ABB RAPID module: MainModule.mod

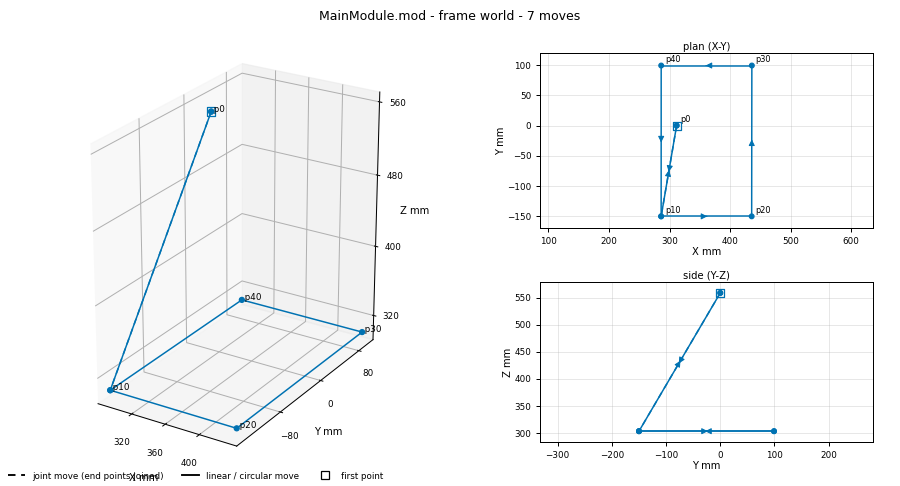
[picture p0: tool path of MainModule.mod in frame world, 7 of 7 moves have a stored position in this frame; points joined in program order, loops and branches not executed]
MODULE MainModule
	CONST robtarget Algus:=[[364.35,0.00,594.00],[0.5,0,0.866025,0],[0,0,0,0],[9E+09,9E+09,9E+09,9E+09,9E+09,9E+09]];
	CONST robtarget p0:=[[311.72,0.00,558.66],[0.0676669,0,0.997708,0],[0,0,0,0],[9E+09,9E+09,9E+09,9E+09,9E+09,9E+09]];
	CONST robtarget p10:=[[286.16,-149.99,303.57],[0.0676667,2.70246E-08,0.997708,1.73496E-07],[-1,0,-1,0],[9E+09,9E+09,9E+09,9E+09,9E+09,9E+09]];
	CONST robtarget p20:=[[435.71,-149.99,303.57],[0.0676665,-1.48195E-07,0.997708,2.84887E-07],[-1,0,-1,0],[9E+09,9E+09,9E+09,9E+09,9E+09,9E+09]];
	CONST robtarget p30:=[[436.00,99.19,303.57],[0.0676668,-2.22625E-07,0.997708,3.78004E-07],[0,-1,0,0],[9E+09,9E+09,9E+09,9E+09,9E+09,9E+09]];
	CONST robtarget p40:=[[286.22,99.19,303.57],[0.0676666,-3.60648E-07,0.997708,3.05387E-07],[0,-1,0,0],[9E+09,9E+09,9E+09,9E+09,9E+09,9E+09]];
	CONST robtarget p50:=[[286.22,99.19,303.57],[0.0676666,-3.60648E-07,0.997708,3.05387E-07],[0,-1,0,0],[9E+09,9E+09,9E+09,9E+09,9E+09,9E+09]];
	TASK PERS tooldata pneumo1:=[TRUE,[[0,0,0],[1,0,0,0]],[-1,[0,0,0],[1,0,0,0],0,0,0]];

    PROC main()
        !MoveJ Algus, v1000, z50, tool0;
        MoveJ p0, v1000, z50, tool0;
        MoveJ p10, v1000, z0, tool0;
        MoveL p20, v1000, z0, tool0;
        MoveL p30, v1000, z0, tool0;
        MoveL p40, v1000, z0, tool0;
        MoveL p10, v1000, z0, tool0;
        MoveL p0, v1000, z50, tool0;
    ENDPROC
ENDMODULE
